DATA_BLOCK "bioPoT.D"
TITLE = Batch I/O Polygon Table Data Block
{ S7_Optimized_Access := 'TRUE' }
AUTHOR : Woermann
VERSION : 1.0
// -- Woermann Automation --
// Date: 2020-06-20
NON_RETAIN
   VAR RETAIN
      PoT : Array[0..15] of "bioPoT.DT";
   END_VAR

BEGIN

END_DATA_BLOCK

